FUNCTION_BLOCK initval_AQ (* a initval for AQ Interface *)
  (* Standard: 61499-2; Description: Copyright (c) 2026 HR Agrartechnik GmbH This program and the accompanying materials are made available under the terms of the Eclipse Public License 2.0 which is available at https://www.eclipse.org/legal/epl-2.0/ SPDX-License-Identifier: EPL-2.0 *)
  (* Version 1.0, 2026-08-13, Franz Höpfinger, HR Agrartechnik GmbH *)
  PACKAGE adapter::types::unidirectional::AQ::initval;
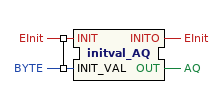
  EVENT_INPUT
    INIT : EInit WITH INIT_VAL; (* Initialization Request *)
  END_EVENT
  EVENT_OUTPUT
    INITO : EInit; (* Initialization Confirm *)
  END_EVENT
  VAR_INPUT
    INIT_VAL : BYTE;
  END_VAR
  PLUGS
    OUT : adapter::types::unidirectional::AQ; (* will output BYTE default at INIT *)
  END_PLUGS
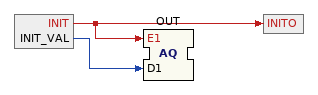
  EVENT_CONNECTIONS
    INIT TO INITO;
    INIT TO OUT.E1;
  END_CONNECTIONS
  DATA_CONNECTIONS
    INIT_VAL TO OUT.D1;
  END_CONNECTIONS
END_FUNCTION_BLOCK
